(* IEC 61131-3 sources: ServoDriveControllerCode_Gen3SOScompressor/src/FB, 18 files *)

(* ---- FB_AnalogInputFilter.st ---- *)
(* ============================================================================
   FB_AnalogInputFilter - Analog Input Filter with Median and Low-Pass

   Project: Gen3 SOS Compressor Servo Controller
   Controller: Yaskawa MP2600iec

   Description:
   Two-stage analog input filter:
   1. Median filter (size 3 or 5) - Removes spike noise and outliers
   2. Low-pass filter (first-order IIR) - Smooths signal, configured by alpha

   The median filter runs first to remove impulsive noise, then the low-pass
   filter smooths the result. This combination is effective for industrial
   analog signals that may have both spike noise and high-frequency interference.

   Low-pass filter implementation:
   - First-order IIR: y[n] = alpha * x[n] + (1-alpha) * y[n-1]
   - Alpha should be calculated by caller: alpha = dt / (tau + dt)
   - Where dt = task cycle time, tau = desired time constant
   - Higher alpha = faster response, less smoothing
   - Lower alpha = slower response, more smoothing

   Configuration:
   - Alpha: Filter coefficient (0.0-1.0), calculated in PRG_Main ST_INIT
   - MedianFilterSize: 3 or 5 samples for median filter
   ============================================================================ *)

FUNCTION_BLOCK FB_AnalogInputFilter
VAR_INPUT
    Enable              : BOOL := TRUE;     (* Enable filtering *)
    RawInput            : INT;              (* Raw analog input (-32768 to +32767) *)
    Alpha               : LREAL;            (* Low-pass filter coefficient (0.0-1.0) *)
    MedianFilterSize    : INT := 3;         (* Median filter size: 3 or 5 *)
END_VAR

VAR_OUTPUT
    FilteredOutput      : INT;              (* Filtered output value *)
    FilteredReal        : LREAL;            (* Filtered output as LREAL *)
    RawReal             : LREAL;            (* Raw input as LREAL *)
END_VAR

VAR
    (* Median filter buffer (size 5, use 3 or 5 based on config) *)
    aMedianBuffer       : ARRAY[0..4] OF LREAL;
    nMedianIndex        : INT := 0;
    aSortBuffer         : ARRAY[0..4] OF LREAL;

    (* Low-pass filter state *)
    rFilteredValue      : LREAL := 0.0;
    rAlpha              : LREAL;

    (* Initialization flag *)
    bInitialized        : BOOL := FALSE;

    (* Temporary variables *)
    i, j                : INT;
    rTemp               : LREAL;
    rMedianResult       : LREAL;
    nSize               : INT;
END_VAR

(* ============================================================================
   Main Logic
   ============================================================================ *)

IF NOT Enable THEN
    (* Pass through raw value when disabled *)
    RawReal := INT_TO_LREAL(RawInput);
    FilteredReal := RawReal;
    FilteredOutput := RawInput;
    RETURN;
END_IF

(* Convert raw input to LREAL *)
RawReal := INT_TO_LREAL(RawInput);

(* Clamp alpha to valid range *)
rAlpha := LIMIT(0.0, Alpha, 1.0);

(* --------------------------------------------------------------------------
   Initialization
   -------------------------------------------------------------------------- *)

IF NOT bInitialized THEN
    (* Fill median buffer with current value *)
    FOR i := 0 TO 4 DO
        aMedianBuffer[i] := RawReal;
    END_FOR
    rFilteredValue := RawReal;
    bInitialized := TRUE;
END_IF

(* --------------------------------------------------------------------------
   Stage 1: Median Filter
   -------------------------------------------------------------------------- *)

(* Limit median size to 3 or 5 *)
IF MedianFilterSize >= 5 THEN
    nSize := 5;
ELSE
    nSize := 3;
END_IF

(* Add new sample to circular buffer *)
aMedianBuffer[nMedianIndex] := RawReal;
nMedianIndex := nMedianIndex + 1;
IF nMedianIndex >= nSize THEN
    nMedianIndex := 0;
END_IF

(* Copy to sort buffer *)
FOR i := 0 TO nSize - 1 DO
    aSortBuffer[i] := aMedianBuffer[i];
END_FOR

(* Simple bubble sort (efficient for small arrays) *)
FOR i := 0 TO nSize - 2 DO
    FOR j := 0 TO nSize - 2 - i DO
        IF aSortBuffer[j] > aSortBuffer[j + 1] THEN
            rTemp := aSortBuffer[j];
            aSortBuffer[j] := aSortBuffer[j + 1];
            aSortBuffer[j + 1] := rTemp;
        END_IF
    END_FOR
END_FOR

(* Get median value (middle element) *)
rMedianResult := aSortBuffer[nSize / 2];

(* --------------------------------------------------------------------------
   Stage 2: Low-Pass Filter (First-Order IIR)
   -------------------------------------------------------------------------- *)

(* Apply low-pass filter: y[n] = alpha * x[n] + (1-alpha) * y[n-1] *)
rFilteredValue := (rAlpha * rMedianResult) + ((1.0 - rAlpha) * rFilteredValue);

(* --------------------------------------------------------------------------
   Output
   -------------------------------------------------------------------------- *)

FilteredReal := rFilteredValue;

(* Convert back to INT with clamping *)
IF rFilteredValue < -32768.0 THEN
    FilteredOutput := -32768;
ELSIF rFilteredValue > 32767.0 THEN
    FilteredOutput := 32767;
ELSE
    FilteredOutput := LREAL_TO_INT(rFilteredValue);
END_IF

END_FUNCTION_BLOCK

(* ---- FB_AnalogProcessor.st ---- *)
(* ============================================================================
   FB_AnalogProcessor - Analog I/O Scaling and Processing

   Project: Gen3 SOS Compressor Servo Controller
   Controller: Yaskawa MP2600iec

   Description:
   Handles scaling of analog input signals for position, velocity, and torque
   reference based on the current operating mode.

   Analog Input Scaling:
   - Raw INT: -32768 to +32767 corresponds to -10V to +10V
   - Scaled to engineering units based on mode and configuration

   Position Mode uses two-stage mapping for consistency with position feedback:
   - Stage 1: In-cylinder region (higher resolution)
   - Stage 2: Out-of-cylinder region (lower resolution)

   Modes:
   - Position (010): Scale to mm using two-stage mapping
   - Velocity (011): Scale to mm/s (linear)
   - Torque (100): Scale to % of rated torque (linear)
   ============================================================================ *)

FUNCTION_BLOCK FB_AnalogProcessor
VAR_INPUT
    Enable              : BOOL;             (* Enable the processor *)
    RawAnalogInput      : INT;              (* Raw analog input value *)
    CurrentMode         : E_OperatingMode;  (* Current operating mode *)

    (* Two-stage position scaling configuration (same as output mapping) *)
    Stage1PosMin        : LREAL;            (* Stage 1 position start (mm) *)
    Stage1PosMax        : LREAL;            (* Stage 1 position end (mm) = transition pos *)
    Stage1VoltMin       : LREAL;            (* Stage 1 voltage start (V) *)
    Stage1VoltMax       : LREAL;            (* Stage 1 voltage end (V) = transition volt *)
    Stage2PosMin        : LREAL;            (* Stage 2 position start (mm) = transition pos *)
    Stage2PosMax        : LREAL;            (* Stage 2 position end (mm) *)
    Stage2VoltMin       : LREAL;            (* Stage 2 voltage start (V) = transition volt *)
    Stage2VoltMax       : LREAL;            (* Stage 2 voltage end (V) *)

    (* Velocity scaling configuration *)
    VelMin              : LREAL;            (* Velocity at -10V (mm/s) *)
    VelMax              : LREAL;            (* Velocity at +10V (mm/s) *)

    (* Torque scaling configuration *)
    TorqueMin           : LREAL;            (* Torque at -10V (%) *)
    TorqueMax           : LREAL;            (* Torque at +10V (%) *)
END_VAR

VAR_OUTPUT
    ScaledPosition      : LREAL;            (* Scaled position reference (mm) *)
    ScaledVelocity      : LREAL;            (* Scaled velocity reference (mm/s) *)
    ScaledTorque        : LREAL;            (* Scaled torque reference (%) *)
    ActiveReference     : LREAL;            (* Currently active reference value *)
    NormalizedInput     : LREAL;            (* Input normalized to 0.0-1.0 range *)
    InputVoltage        : LREAL;            (* Calculated input voltage (-10 to +10) *)
    InStage1            : BOOL;             (* Position input is in stage 1 region *)
    InStage2            : BOOL;             (* Position input is in stage 2 region *)
END_VAR

VAR
    rNormalized         : LREAL;            (* Normalized value 0.0 to 1.0 *)
    rStageNormalized    : LREAL;            (* Normalized value within stage *)
END_VAR

(* ============================================================================
   Constants
   ============================================================================ *)
VAR CONSTANT
    RAW_MIN             : LREAL := -32768.0;    (* Minimum raw value *)
    RAW_MAX             : LREAL := 32767.0;     (* Maximum raw value *)
    RAW_RANGE           : LREAL := 65535.0;     (* Total raw range *)
    VOLT_MIN            : LREAL := -10.0;       (* Minimum voltage *)
    VOLT_MAX            : LREAL := 10.0;        (* Maximum voltage *)
    VOLT_RANGE          : LREAL := 20.0;        (* Total voltage range *)
END_VAR

(* ============================================================================
   Main Logic
   ============================================================================ *)

IF NOT Enable THEN
    ScaledPosition := 0.0;
    ScaledVelocity := 0.0;
    ScaledTorque := 0.0;
    ActiveReference := 0.0;
    NormalizedInput := 0.5;
    InputVoltage := 0.0;
    InStage1 := FALSE;
    InStage2 := FALSE;
    RETURN;
END_IF

(* Normalize raw input to 0.0-1.0 range *)
rNormalized := (INT_TO_LREAL(RawAnalogInput) - RAW_MIN) / RAW_RANGE;
NormalizedInput := rNormalized;

(* Calculate input voltage *)
InputVoltage := VOLT_MIN + (rNormalized * VOLT_RANGE);

(* Scale velocity and torque (simple linear mapping) *)
ScaledVelocity := VelMin + (rNormalized * (VelMax - VelMin));
ScaledTorque := TorqueMin + (rNormalized * (TorqueMax - TorqueMin));

(* Scale position using two-stage mapping (inverse of FB_PositionMapping) *)
(* Determine which stage based on input voltage *)
(* Use < (not <=) so boundary value is handled by stage 2 only *)
IF InputVoltage < Stage1VoltMax THEN
    (* Stage 1: In-cylinder region *)
    InStage1 := TRUE;
    InStage2 := FALSE;

    (* Calculate normalized position within stage 1 *)
    IF (Stage1VoltMax - Stage1VoltMin) > 0.0 THEN
        rStageNormalized := (InputVoltage - Stage1VoltMin) / (Stage1VoltMax - Stage1VoltMin);
    ELSE
        rStageNormalized := 0.0;
    END_IF

    (* Clamp to 0.0-1.0 range *)
    rStageNormalized := LIMIT(0.0, rStageNormalized, 1.0);

    (* Calculate position for stage 1 *)
    ScaledPosition := Stage1PosMin + (rStageNormalized * (Stage1PosMax - Stage1PosMin));

ELSE
    (* Stage 2: Out-of-cylinder region *)
    InStage1 := FALSE;
    InStage2 := TRUE;

    (* Calculate normalized position within stage 2 *)
    IF (Stage2VoltMax - Stage2VoltMin) > 0.0 THEN
        rStageNormalized := (InputVoltage - Stage2VoltMin) / (Stage2VoltMax - Stage2VoltMin);
    ELSE
        rStageNormalized := 0.0;
    END_IF

    (* Clamp to 0.0-1.0 range *)
    rStageNormalized := LIMIT(0.0, rStageNormalized, 1.0);

    (* Calculate position for stage 2 *)
    ScaledPosition := Stage2PosMin + (rStageNormalized * (Stage2PosMax - Stage2PosMin));
END_IF

(* Select active reference based on mode *)
CASE CurrentMode OF
    MODE_POSITION:
        ActiveReference := ScaledPosition;

    MODE_VELOCITY:
        ActiveReference := ScaledVelocity;

    MODE_TORQUE:
        ActiveReference := ScaledTorque;

ELSE
    ActiveReference := 0.0;
END_CASE

END_FUNCTION_BLOCK

(* ---- FB_DigitalInputFilter.st ---- *)
(* ============================================================================
   FB_DigitalInputFilter - Digital Input Debounce Filter

   Project: Gen3 SOS Compressor Servo Controller
   Controller: Yaskawa MP2600iec

   Description:
   Debounces a digital input signal by requiring the input to be stable for
   a configurable time before the output changes.

   Features:
   - Configurable debounce time
   - Edge detection outputs
   - Raw input passthrough for debugging
   ============================================================================ *)

FUNCTION_BLOCK FB_DigitalInputFilter
VAR_INPUT
    RawInput            : BOOL;             (* Raw digital input *)
    DebounceTime        : TIME := T#10MS;   (* Debounce time *)
END_VAR

VAR_OUTPUT
    FilteredOutput      : BOOL;             (* Debounced output *)
    RisingEdge          : BOOL;             (* Rising edge detected on filtered output *)
    FallingEdge         : BOOL;             (* Falling edge detected on filtered output *)
    Stable              : BOOL;             (* Output has been stable (not changing) *)
    RawPassthrough      : BOOL;             (* Raw input passthrough for debugging *)
END_VAR

VAR
    tDebounce           : TON;              (* Debounce timer *)
    bLastRaw            : BOOL;             (* Previous raw input state *)
    bLastFiltered       : BOOL;             (* Previous filtered output state *)
    bPendingState       : BOOL;             (* State we're debouncing toward *)
    bFirstScan          : BOOL := TRUE;     (* First scan flag for initialization *)
END_VAR

(* ============================================================================
   Main Logic
   ============================================================================ *)

(* Passthrough for debugging *)
RawPassthrough := RawInput;

(* First scan initialization - accept current input state immediately *)
IF bFirstScan THEN
    FilteredOutput := RawInput;
    bLastRaw := RawInput;
    bLastFiltered := RawInput;
    bPendingState := RawInput;
    Stable := TRUE;
    RisingEdge := FALSE;
    FallingEdge := FALSE;
    bFirstScan := FALSE;
    RETURN;
END_IF

(* Detect raw input change *)
IF RawInput <> bLastRaw THEN
    (* Input changed - start debouncing toward new state *)
    bPendingState := RawInput;
    tDebounce(IN := FALSE);  (* Reset timer *)
END_IF

bLastRaw := RawInput;

(* Run debounce timer if pending state differs from current output *)
IF bPendingState <> FilteredOutput THEN
    tDebounce(IN := TRUE, PT := DebounceTime);
    Stable := FALSE;

    IF tDebounce.Q THEN
        (* Debounce complete - update output *)
        FilteredOutput := bPendingState;
        tDebounce(IN := FALSE);
        Stable := TRUE;
    END_IF
ELSE
    (* No state change pending *)
    tDebounce(IN := FALSE);
    Stable := TRUE;
END_IF

(* Edge detection on filtered output *)
RisingEdge := FilteredOutput AND NOT bLastFiltered;
FallingEdge := NOT FilteredOutput AND bLastFiltered;
bLastFiltered := FilteredOutput;

END_FUNCTION_BLOCK

(* ---- FB_EncoderManager.st ---- *)
(* ============================================================================
   FB_EncoderManager - Absolute Encoder Validation Manager

   Project: Gen3 SOS Compressor Servo Controller
   Controller: Yaskawa MP2600iec

   Description:
   Validates absolute encoder status on startup using Yaskawa's
   AbsolutePositionManager function block. Determines if homing is required
   due to encoder battery failure or multi-turn data corruption.

   The Sigma-7 absolute encoder maintains position across power cycles via
   battery backup. If the battery fails or multi-turn data is corrupted,
   the encoder position is invalid and homing is required.

   States:
   - IDLE: Waiting for check trigger
   - CHECK_INIT: Initialize AbsolutePositionManager
   - CHECK_STATUS: Query encoder status
   - COMPLETE: Check finished, outputs valid
   - ERROR: Error during check

   Integration:
   - Called from ST_ENCODER_CHECK state in PRG_Main
   - Sets AbsHomeRequired output if encoder invalid
   - PRG_Main uses this to set flagAbsHomeRequired
   ============================================================================ *)

FUNCTION_BLOCK FB_EncoderManager
VAR_INPUT
    Enable              : BOOL;             (* Enable the function block *)
    Axis                : AXIS_REF;         (* PLCopen axis reference *)
    CheckOnStartup      : BOOL;             (* Trigger startup check *)
END_VAR

VAR_OUTPUT
    EncoderValid        : BOOL;             (* Absolute position is valid *)
    BatteryOK           : BOOL;             (* Encoder battery status OK *)
    MultiTurnValid      : BOOL;             (* Multi-turn counter data valid *)
    AbsHomeRequired     : BOOL;             (* Homing required due to encoder issue *)
    CheckComplete       : BOOL;             (* Startup check finished *)
    Busy                : BOOL;             (* Check in progress *)
    Error               : BOOL;             (* Error occurred during check *)
    ErrorID             : DWORD;            (* Error code if Error=TRUE *)
END_VAR

VAR
    (* Yaskawa AbsolutePositionManager function block *)
    fbAbsPosManager     : AbsolutePositionManager;

    (* State machine *)
    eState              : INT := ENC_IDLE;

    (* Edge detection *)
    rTrigCheck          : R_TRIG;

    (* Timeout *)
    tCheckTimeout       : TON;

    (* Internal status *)
    bCheckTriggered     : BOOL;
END_VAR

(* ============================================================================
   Constants
   ============================================================================ *)
VAR CONSTANT
    ENC_IDLE            : INT := 0;         (* Idle state *)
    ENC_CHECK_INIT      : INT := 1;         (* Initialize check *)
    ENC_CHECK_STATUS    : INT := 2;         (* Query status *)
    ENC_COMPLETE        : INT := 3;         (* Check complete *)
    ENC_ERROR           : INT := 4;         (* Error state *)

    CHECK_TIMEOUT       : TIME := T#2S;     (* Timeout for encoder check *)
END_VAR

(* ============================================================================
   Main Logic
   ============================================================================ *)

IF NOT Enable THEN
    (* Reset all outputs when disabled *)
    EncoderValid := FALSE;
    BatteryOK := FALSE;
    MultiTurnValid := FALSE;
    AbsHomeRequired := FALSE;
    CheckComplete := FALSE;
    Busy := FALSE;
    Error := FALSE;
    ErrorID := 0;
    eState := ENC_IDLE;
    tCheckTimeout(IN := FALSE);
    fbAbsPosManager(Enable := FALSE);
    RETURN;
END_IF

(* Detect rising edge on CheckOnStartup *)
rTrigCheck(CLK := CheckOnStartup);

CASE eState OF

    ENC_IDLE:
        (* Waiting for check trigger *)
        Busy := FALSE;
        CheckComplete := FALSE;

        IF rTrigCheck.Q OR (CheckOnStartup AND NOT bCheckTriggered) THEN
            bCheckTriggered := TRUE;
            Busy := TRUE;
            Error := FALSE;
            ErrorID := 0;
            tCheckTimeout(IN := FALSE);
            eState := ENC_CHECK_INIT;
        END_IF

    ENC_CHECK_INIT:
        (* Initialize AbsolutePositionManager *)
        (* Start timeout timer *)
        tCheckTimeout(IN := TRUE, PT := CHECK_TIMEOUT);

        (* Enable the AbsolutePositionManager *)
        fbAbsPosManager(
            Axis := Axis,
            Enable := TRUE
        );

        (* Wait for FB to initialize or check for immediate status *)
        IF fbAbsPosManager.Valid THEN
            eState := ENC_CHECK_STATUS;
        ELSIF fbAbsPosManager.Error THEN
            Error := TRUE;
            ErrorID := fbAbsPosManager.ErrorID;
            eState := ENC_ERROR;
        ELSIF tCheckTimeout.Q THEN
            Error := TRUE;
            ErrorID := 16#8001;  (* Timeout error code *)
            eState := ENC_ERROR;
        END_IF

    ENC_CHECK_STATUS:
        (* Query encoder status from AbsolutePositionManager *)
        fbAbsPosManager(
            Axis := Axis,
            Enable := TRUE
        );

        (* Read status outputs *)
        (* Note: Actual output names depend on Yaskawa's AbsolutePositionManager interface *)
        (* Common outputs: AbsolutePositionValid, BatteryStatus, etc. *)

        (* Check for valid absolute position *)
        IF fbAbsPosManager.Valid THEN
            (* Evaluate encoder health *)
            (* AbsolutePositionManager typically provides:
               - Valid: Overall validity
               - AbsolutePositionValid: Position data is valid
               - BatteryAlarm: Battery has failed or is low
               - MultiTurnOverflow: Multi-turn counter overflow *)

            (* For Sigma-7, check if position is valid and no alarms *)
            EncoderValid := fbAbsPosManager.AbsolutePositionValid;
            BatteryOK := NOT fbAbsPosManager.BatteryAlarm;
            MultiTurnValid := NOT fbAbsPosManager.MultiTurnOverflow;

            (* Homing required if any issue detected *)
            AbsHomeRequired := NOT EncoderValid OR
                               NOT BatteryOK OR
                               NOT MultiTurnValid;

            CheckComplete := TRUE;
            Busy := FALSE;
            tCheckTimeout(IN := FALSE);
            eState := ENC_COMPLETE;

        ELSIF fbAbsPosManager.Error THEN
            Error := TRUE;
            ErrorID := fbAbsPosManager.ErrorID;
            eState := ENC_ERROR;

        ELSIF tCheckTimeout.Q THEN
            Error := TRUE;
            ErrorID := 16#8001;  (* Timeout error code *)
            eState := ENC_ERROR;
        END_IF

    ENC_COMPLETE:
        (* Check complete - hold outputs until disabled or new check *)
        Busy := FALSE;
        CheckComplete := TRUE;

        (* Allow re-check if CheckOnStartup toggled *)
        IF NOT CheckOnStartup THEN
            bCheckTriggered := FALSE;
        END_IF

        IF rTrigCheck.Q THEN
            (* New check requested *)
            CheckComplete := FALSE;
            Busy := TRUE;
            tCheckTimeout(IN := FALSE);
            eState := ENC_CHECK_INIT;
        END_IF

    ENC_ERROR:
        (* Error state *)
        Busy := FALSE;
        CheckComplete := FALSE;

        (* Assume encoder invalid on error - safe default *)
        EncoderValid := FALSE;
        BatteryOK := FALSE;
        MultiTurnValid := FALSE;
        AbsHomeRequired := TRUE;

        (* Disable the AbsolutePositionManager *)
        fbAbsPosManager(Enable := FALSE);
        tCheckTimeout(IN := FALSE);

        (* Allow retry if CheckOnStartup toggled *)
        IF NOT CheckOnStartup THEN
            bCheckTriggered := FALSE;
            Error := FALSE;
            ErrorID := 0;
            eState := ENC_IDLE;
        END_IF

END_CASE

END_FUNCTION_BLOCK

(* ---- FB_GoHome.st ---- *)
(* ============================================================================
   FB_GoHome - Go Home Mode Handler (Mode 101)

   Project: Gen3 SOS Compressor Servo Controller
   Controller: Yaskawa MP2600iec

   Description:
   Handles Mode 101 (Go Home) which moves the axis to the home position
   (at the home limit switch). This mode checks homing requirements before
   executing and redirects to homing mode if needed.

   Behavior:
   - If AbsHomeRequired is TRUE: Set RedirectToHoming, PRG_Main switches to 110
   - If requirements met: Execute MC_MoveAbsolute to HomePosition
   - After reaching position: Hold there until mode change

   Note: EOTHomeRequired does NOT block Go Home - the axis can still move
   to the home position even if EOT homing hasn't been done. Only
   AbsHomeRequired (encoder validity) blocks the move.

   Integration:
   - Called from ST_GO_HOME state in PRG_Main
   - RedirectToHoming signals PRG_Main to switch to ST_HOME_LIMIT
   - Abort input for motion enable drop handling
   ============================================================================ *)

FUNCTION_BLOCK FB_GoHome
VAR_INPUT
    Enable              : BOOL;             (* Enable the function block *)
    Execute             : BOOL;             (* Start go home sequence *)
    Axis                : AXIS_REF;         (* PLCopen axis reference *)

    (* Homing requirement flags *)
    AbsHomeRequired     : BOOL;             (* Encoder homing required (blocks Go Home) *)
    EOTHomeRequired     : BOOL;             (* EOT homing required (does NOT block) *)

    (* Configuration *)
    HomePosition        : LREAL;            (* Target home position (mm) *)
    HomeVelocity        : LREAL;            (* Movement velocity (mm/s) *)

    (* Control *)
    Abort               : BOOL;             (* Abort the move *)
END_VAR

VAR_OUTPUT
    Active              : BOOL;             (* Sequence is running *)
    Done                : BOOL;             (* At home position *)
    AtPosition          : BOOL;             (* Currently at home position *)
    HomingRequired      : BOOL;             (* Homing must be done first *)
    RedirectToHoming    : BOOL;             (* Caller should switch to homing mode *)
    InMotion            : BOOL;             (* Currently moving *)
    Error               : BOOL;             (* Error occurred *)
    ErrorID             : DWORD;            (* Error code if Error=TRUE *)
END_VAR

VAR
    (* PLCopen function blocks *)
    fbMoveAbsolute      : MC_MoveAbsolute;
    fbHalt              : MC_Halt;

    (* State machine *)
    eState              : INT := GOH_IDLE;

    (* Edge detection *)
    rTrigExecute        : R_TRIG;

    (* Position tolerance for "at position" detection *)
    rPosTolerance       : LREAL := 0.1;     (* mm *)
END_VAR

(* ============================================================================
   Constants
   ============================================================================ *)
VAR CONSTANT
    GOH_IDLE            : INT := 0;         (* Idle state *)
    GOH_CHECK_REQ       : INT := 1;         (* Check requirements *)
    GOH_REDIRECT        : INT := 2;         (* Redirect to homing *)
    GOH_MOVING          : INT := 3;         (* Moving to home *)
    GOH_AT_POSITION     : INT := 4;         (* At home position *)
    GOH_ABORTING        : INT := 5;         (* Aborting move *)
    GOH_ERROR           : INT := 6;         (* Error state *)
END_VAR

(* ============================================================================
   Main Logic
   ============================================================================ *)

IF NOT Enable THEN
    (* Reset all outputs when disabled *)
    Active := FALSE;
    Done := FALSE;
    AtPosition := FALSE;
    HomingRequired := FALSE;
    RedirectToHoming := FALSE;
    InMotion := FALSE;
    Error := FALSE;
    ErrorID := 0;
    eState := GOH_IDLE;
    fbMoveAbsolute(Execute := FALSE);
    fbHalt(Execute := FALSE);
    RETURN;
END_IF

(* Detect rising edge on Execute *)
rTrigExecute(CLK := Execute);

(* Handle abort in any state *)
IF Abort AND (eState <> GOH_IDLE) AND (eState <> GOH_ERROR) AND (eState <> GOH_REDIRECT) THEN
    fbMoveAbsolute(Execute := FALSE);
    eState := GOH_ABORTING;
END_IF

CASE eState OF

    GOH_IDLE:
        (* Waiting for execute command *)
        Active := FALSE;
        Done := FALSE;
        AtPosition := FALSE;
        HomingRequired := FALSE;
        RedirectToHoming := FALSE;
        InMotion := FALSE;
        Error := FALSE;
        ErrorID := 0;

        (* Reset function blocks *)
        fbMoveAbsolute(Execute := FALSE);
        fbHalt(Execute := FALSE);

        IF rTrigExecute.Q OR Execute THEN
            Active := TRUE;
            eState := GOH_CHECK_REQ;
        END_IF

    GOH_CHECK_REQ:
        (* Check homing requirements *)

        IF AbsHomeRequired THEN
            (* Encoder homing required - cannot go home without valid position *)
            HomingRequired := TRUE;
            RedirectToHoming := TRUE;
            eState := GOH_REDIRECT;

        ELSE
            (* Requirements met (or only EOT homing needed) - proceed with move *)
            HomingRequired := FALSE;
            RedirectToHoming := FALSE;
            eState := GOH_MOVING;
        END_IF

    GOH_REDIRECT:
        (* Waiting for PRG_Main to handle redirect *)
        (* Stay in this state - PRG_Main will transition to ST_HOME_LIMIT *)
        (* This FB will be disabled when state changes *)
        Active := TRUE;
        HomingRequired := TRUE;
        RedirectToHoming := TRUE;

    GOH_MOVING:
        (* Execute move to home position *)
        fbMoveAbsolute(
            Axis := Axis,
            Execute := TRUE,
            Position := HomePosition,
            Velocity := HomeVelocity,
            Acceleration := 0.0,    (* Use axis default *)
            Deceleration := 0.0,    (* Use axis default *)
            Jerk := 0.0             (* Use axis default *)
        );

        InMotion := fbMoveAbsolute.Busy;

        IF fbMoveAbsolute.Done THEN
            (* Move complete - reset FB for next use
               NOTE: Setting Execute := FALSE does NOT release position control.
               Per PLCopen standard, axis remains in "Standstill" state with
               active servo position holding. This is standard practice. *)
            fbMoveAbsolute(Execute := FALSE);
            Done := TRUE;
            AtPosition := TRUE;
            InMotion := FALSE;
            eState := GOH_AT_POSITION;

        ELSIF fbMoveAbsolute.Error THEN
            (* Move failed *)
            Error := TRUE;
            ErrorID := fbMoveAbsolute.ErrorID;
            fbMoveAbsolute(Execute := FALSE);
            eState := GOH_ERROR;

        ELSIF fbMoveAbsolute.CommandAborted THEN
            (* Move was aborted externally *)
            fbMoveAbsolute(Execute := FALSE);
            eState := GOH_ABORTING;
        END_IF

    GOH_AT_POSITION:
        (* At home position - hold here until mode change *)
        Done := TRUE;
        AtPosition := TRUE;
        InMotion := FALSE;
        Active := TRUE;

        (* Check if still at position (could drift in some cases) *)
        (* Note: In practice, the drive holds position in servo mode *)

        (* If Execute goes low, we can reset for next time *)
        IF NOT Execute THEN
            Done := FALSE;
            eState := GOH_IDLE;
        END_IF

    GOH_ABORTING:
        (* Aborting move - execute halt *)
        fbHalt(
            Axis := Axis,
            Execute := TRUE
        );

        IF fbHalt.Done THEN
            fbHalt(Execute := FALSE);
            Active := FALSE;
            InMotion := FALSE;
            eState := GOH_IDLE;

        ELSIF fbHalt.Error THEN
            (* Halt failed - still try to go to idle *)
            fbHalt(Execute := FALSE);
            eState := GOH_ERROR;
        END_IF

    GOH_ERROR:
        (* Error state *)
        Active := FALSE;
        InMotion := FALSE;
        Done := FALSE;

        (* Allow reset when Execute goes low *)
        IF NOT Execute THEN
            Error := FALSE;
            ErrorID := 0;
            eState := GOH_IDLE;
        END_IF

END_CASE

END_FUNCTION_BLOCK

(* ---- FB_HandshakeManager.st ---- *)
(* ============================================================================
   FB_HandshakeManager - Master-Slave Handshake Manager

   Project: Gen3 SOS Compressor Servo Controller
   Controller: Yaskawa MP2600iec

   Description:
   Manages the handshake protocol between master and slave for:
   1. Mode entry handshake: 3-bit mode command/confirmation with timeout
   2. Fault reset handshake: FaultReset HIGH + MotionEnable LOW + fault mirroring

   Mode Entry Handshake Sequence:
   1. Master sets mode bits (DI0-2)
   2. Slave decodes and validates mode
   3. Slave sets confirmation bits (DO0-2) to match
   4. Master sets diMotionEnable HIGH
   5. Slave verifies mode bits still match → handshake complete
   6. If timeout or mismatch → handshake failed

   Fault Reset Handshake (with fault code mirroring):
   1. Slave is in fault state with doFaultActive = HIGH
   2. Slave outputs fault code on DO0-DO2
   3. Master reads fault code and sets DI0-DI2 to mirror it
   4. Master sets diFaultReset HIGH while diMotionEnable = LOW
   5. Slave verifies DI0-DI2 matches fault code (level-based, not edge)
   6. FaultResetValid goes TRUE, caller clears fault
   7. Master sees fault cleared, releases diFaultReset

   NOTE: All inputs should be pre-filtered/debounced by the caller.
   ============================================================================ *)

FUNCTION_BLOCK FB_HandshakeManager
VAR_INPUT
    Enable              : BOOL;             (* Enable handshake manager *)

    (* Mode handshake inputs *)
    RequestedMode       : E_OperatingMode;  (* Mode requested by master *)
    ModeStable          : BOOL;             (* Mode inputs are stable *)
    MotionEnable        : BOOL;             (* Motion enable from master - should be filtered *)

    (* Fault reset inputs *)
    FaultReset          : BOOL;             (* Fault reset signal from master - should be filtered *)
    InFaultState        : BOOL;             (* Currently in fault state *)
    ActiveFaultCode     : E_FaultCode;      (* Active fault code for mirroring check *)

    (* Configuration *)
    HandshakeTimeout    : TIME := T#500MS;  (* Timeout for handshake *)
END_VAR

VAR_OUTPUT
    (* Mode handshake outputs *)
    ConfirmedMode       : E_OperatingMode;  (* Current confirmed mode (valid when HandshakeComplete) *)
    HandshakeActive     : BOOL;             (* TRUE from handshake start until complete/timeout *)
    HandshakeComplete   : BOOL;             (* TRUE when handshake succeeded (persists until MotionEnable drops) *)
    HandshakeTimeout_Q  : BOOL;             (* TRUE when timeout occurred (persists until MotionEnable drops) *)

    (* Confirmation bits for digital outputs *)
    ConfirmBit0         : BOOL;             (* DO0 value *)
    ConfirmBit1         : BOOL;             (* DO1 value *)
    ConfirmBit2         : BOOL;             (* DO2 value *)

    (* Fault reset outputs *)
    FaultResetEdge      : BOOL;             (* Fault reset rising edge detected (single scan pulse) *)
    FaultResetValid     : BOOL;             (* Fault reset conditions met (level-based, stays TRUE while valid) *)
END_VAR

VAR
    (* State machine *)
    eState              : INT := HS_IDLE;   (* Handshake state - initialized to HS_IDLE *)

    (* Timers *)
    tTimeout            : TON;              (* Handshake timeout timer *)

    (* Edge detection *)
    rTrigFaultReset     : R_TRIG;           (* Rising edge on fault reset *)

    (* Internal tracking *)
    eModeAtStart        : E_OperatingMode;  (* Mode when handshake started *)
    bModeStableAtStart  : BOOL;             (* Capture mode stability at handshake start *)
END_VAR

(* ============================================================================
   Constants for state machine
   ============================================================================ *)
VAR CONSTANT
    HS_IDLE             : INT := 0;         (* Idle, no handshake active *)
    HS_WAIT_MOTION_EN   : INT := 1;         (* Waiting for motion enable *)
    HS_VERIFY_MODE      : INT := 2;         (* Verifying mode match *)
    HS_COMPLETE         : INT := 3;         (* Handshake complete *)
    HS_TIMEOUT          : INT := 4;         (* Handshake timed out *)
END_VAR

(* ============================================================================
   Main Logic
   ============================================================================ *)

IF NOT Enable THEN
    (* Reset all outputs when disabled *)
    ConfirmedMode := MODE_IDLE;
    HandshakeActive := FALSE;
    HandshakeComplete := FALSE;
    HandshakeTimeout_Q := FALSE;
    ConfirmBit0 := FALSE;
    ConfirmBit1 := FALSE;
    ConfirmBit2 := FALSE;
    FaultResetEdge := FALSE;
    FaultResetValid := FALSE;
    eState := HS_IDLE;
    tTimeout(IN := FALSE);
    RETURN;
END_IF

(* --------------------------------------------------------------------------
   Fault Reset Handshake Detection (with fault code mirroring)
   Uses LEVEL-based detection to avoid race conditions.
   The caller should detect the rising edge of FaultResetValid if needed.
   -------------------------------------------------------------------------- *)
rTrigFaultReset(CLK := FaultReset);
FaultResetEdge := rTrigFaultReset.Q;

(* Fault reset is valid when ALL conditions are met (level-based):
   - FaultReset is HIGH (level, not edge)
   - MotionEnable is LOW
   - We are in fault state
   - Active fault code is not FAULT_NONE
   - Master has mirrored the fault code on DI0-2 (RequestedMode matches ActiveFaultCode) *)
FaultResetValid := FaultReset AND
                   (NOT MotionEnable) AND
                   InFaultState AND
                   (ActiveFaultCode <> FAULT_NONE) AND
                   FaultMatchesModeBits(ActiveFaultCode, RequestedMode);

(* --------------------------------------------------------------------------
   Mode Handshake State Machine
   -------------------------------------------------------------------------- *)
CASE eState OF

    HS_IDLE:
        (* Reset outputs *)
        HandshakeActive := FALSE;
        HandshakeComplete := FALSE;
        HandshakeTimeout_Q := FALSE;
        tTimeout(IN := FALSE);

        (* Start handshake when mode is stable and different from idle
           (or when transitioning to a new mode) *)
        IF ModeStable AND (RequestedMode <> MODE_IDLE) AND NOT MotionEnable THEN
            (* Set confirmation to match requested mode *)
            ConfirmedMode := RequestedMode;
            SetConfirmBits(RequestedMode);
            eModeAtStart := RequestedMode;
            bModeStableAtStart := TRUE;
            HandshakeActive := TRUE;
            eState := HS_WAIT_MOTION_EN;
            tTimeout(IN := TRUE, PT := HandshakeTimeout);
        ELSIF ModeStable AND (RequestedMode = MODE_IDLE) THEN
            (* Idle mode - just confirm it *)
            ConfirmedMode := MODE_IDLE;
            SetConfirmBits(MODE_IDLE);
        END_IF

    HS_WAIT_MOTION_EN:
        (* Waiting for master to assert motion enable *)
        (* Timer must be called each scan to update *)
        tTimeout(IN := TRUE, PT := HandshakeTimeout);

        IF tTimeout.Q THEN
            (* Timeout - handshake failed *)
            tTimeout(IN := FALSE);
            eState := HS_TIMEOUT;

        ELSIF RequestedMode <> eModeAtStart THEN
            (* Mode changed during handshake - abort and reset timer *)
            tTimeout(IN := FALSE);
            eState := HS_IDLE;

        ELSIF MotionEnable THEN
            (* Motion enable received, verify mode still matches *)
            eState := HS_VERIFY_MODE;
        END_IF

    HS_VERIFY_MODE:
        (* Verify requested mode hasn't changed since handshake start *)
        IF RequestedMode = eModeAtStart THEN
            (* Mode matches - handshake complete *)
            HandshakeComplete := TRUE;
            HandshakeActive := FALSE;
            tTimeout(IN := FALSE);
            eState := HS_COMPLETE;
        ELSE
            (* Mismatch - treat as timeout/failure *)
            tTimeout(IN := FALSE);
            eState := HS_TIMEOUT;
        END_IF

    HS_COMPLETE:
        (* Handshake complete - stay here until motion enable drops *)
        IF NOT MotionEnable THEN
            (* Motion disabled - return to idle *)
            HandshakeComplete := FALSE;
            eState := HS_IDLE;
        END_IF

    HS_TIMEOUT:
        (* Handshake timed out or failed *)
        HandshakeTimeout_Q := TRUE;
        HandshakeActive := FALSE;
        ConfirmedMode := MODE_IDLE;  (* Reset confirmed mode on failure *)
        SetConfirmBits(MODE_IDLE);
        tTimeout(IN := FALSE);

        (* Exit timeout when motion enable drops - simpler and more reliable *)
        IF NOT MotionEnable THEN
            HandshakeTimeout_Q := FALSE;
            eState := HS_IDLE;
        END_IF

END_CASE

END_FUNCTION_BLOCK

(* ============================================================================
   Helper Method: Set Confirmation Bits from Mode
   Uses centralized conversion functions from EnumConversions.st
   ============================================================================ *)
METHOD PRIVATE SetConfirmBits
VAR_INPUT
    Mode : E_OperatingMode;
END_VAR

(* Use centralized ModeToBits function *)
ModeToBits(Mode, ConfirmBit0, ConfirmBit1, ConfirmBit2);

END_METHOD

(* ---- FB_HomeEOT.st ---- *)
(* ============================================================================
   FB_HomeEOT - End-of-Travel Homing Sequence Handler (Mode 111)

   Project: Gen3 SOS Compressor Servo Controller
   Controller: Yaskawa MP2600iec

   Description:
   Encapsulates the complete End-of-Travel (EOT) homing sequence for Mode 111.
   Uses torque-limited velocity control to find the mechanical end stop, then
   calculates a coordinate offset for master/slave translation.

   Sequence:
   1. CHECK_REQ: Verify AbsHomeRequired is FALSE (limit switch homing must be done first)
   2. FAST_APPROACH: Fast jog toward EOT with torque limiting for safety
   3. SLOW_APPROACH: Slow torque-limited approach when near expected position
   4. STALL_DETECT: Confirm stall condition (velocity near zero, torque at limit)
   5. SETREF: Calculate coordinate offset (preserves encoder zero from Mode 110)

   Coordinate System:
   This FB calculates EOTOffset for master/slave coordinate transformation:
   - Master position = Slave position + EOTOffset
   - EOTOffset = ExpectedEOTPosition - ActualEOTPosition (encoder value at stall)

   This preserves the limit switch zero reference from Mode 110 while allowing
   the master to see the expected position value at EOT.

   Uses Y_DirectControl:
   - Mode 2 (velocity mode) with torque limiting for safe mechanical contact

   Integration:
   - Called from ST_HOME_EOT state in PRG_Main
   - RequiresLimitHome output signals need for Mode 110 first
   - Abort input for motion enable drop handling
   ============================================================================ *)

FUNCTION_BLOCK FB_HomeEOT
VAR_INPUT
    Enable              : BOOL;             (* Enable the function block *)
    Execute             : BOOL;             (* Start homing sequence *)
    Axis                : AXIS_REF;         (* PLCopen axis reference *)

    (* Homing requirement check *)
    AbsHomeRequired     : BOOL;             (* Limit switch homing required (blocks EOT homing) *)

    (* Configuration *)
    FastVelocity        : LREAL;            (* Fast approach velocity (mm/s) *)
    SlowVelocity        : LREAL;            (* Slow approach velocity (mm/s) *)
    TorqueLimit         : LREAL;            (* Torque limit during approach (%) *)
    TorqueThreshold     : LREAL;            (* Torque threshold for stall detection (%) *)
    ApproachDistance    : LREAL;            (* Distance before EOT to switch to slow (mm) *)
    ExpectedEOTPosition : LREAL;            (* Expected position at EOT (mm) *)
    StallDetectTime     : TIME;             (* Time to confirm stall condition *)
    Timeout             : TIME;             (* Overall sequence timeout *)

    (* Feedback inputs *)
    ActualPosition      : LREAL;            (* Current position (mm) *)
    ActualVelocity      : LREAL;            (* Current velocity (mm/s) *)
    ActualTorque        : LREAL;            (* Current torque (% of rated) *)

    (* Control *)
    Abort               : BOOL;             (* Abort the sequence *)
END_VAR

VAR_OUTPUT
    Active              : BOOL;             (* Sequence is running *)
    Done                : BOOL;             (* Homing complete *)
    InMotion            : BOOL;             (* Currently moving *)
    Error               : BOOL;             (* Error occurred *)
    ErrorID             : DWORD;            (* Error code if Error=TRUE *)
    RequiresLimitHome   : BOOL;             (* Must do limit switch homing first *)
    EOTPosition         : LREAL;            (* Recorded encoder position at EOT stall *)
    EOTOffset           : LREAL;            (* Calculated coordinate offset *)
END_VAR

VAR
    (* Yaskawa function blocks *)
    fbDirectControl     : Y_DirectControl;
    fbHalt              : MC_Halt;

    (* State machine *)
    eState              : INT := HE_IDLE;

    (* Edge detection *)
    rTrigExecute        : R_TRIG;

    (* Timers *)
    tTimeout            : TON;              (* Overall timeout *)
    tStallConfirm       : TON;              (* Stall confirmation timer *)

    (* Stall detection threshold with hysteresis *)
    rVelocityThreshold  : LREAL := 0.5;     (* mm/s - velocity considered "stopped" *)
    rTorqueMultiplier   : LREAL := 0.9;     (* Multiplier for torque threshold *)
END_VAR

(* ============================================================================
   Constants
   ============================================================================ *)
VAR CONSTANT
    HE_IDLE             : INT := 0;         (* Idle state *)
    HE_CHECK_REQ        : INT := 1;         (* Check requirements *)
    HE_REQUIRES_HOME    : INT := 2;         (* Limit homing required first *)
    HE_FAST_APPROACH    : INT := 3;         (* Fast approach to near EOT *)
    HE_SLOW_APPROACH    : INT := 4;         (* Slow torque-limited approach *)
    HE_STALL_DETECT     : INT := 5;         (* Confirming stall condition *)
    HE_SETREF           : INT := 6;         (* Calculate offset *)
    HE_DONE             : INT := 7;         (* Sequence complete *)
    HE_ABORTING         : INT := 8;         (* Aborting sequence *)
    HE_ERROR            : INT := 9;         (* Error state *)

    (* Error codes *)
    ERR_TIMEOUT         : DWORD := 16#8011; (* Homing timeout *)
    ERR_DRIVE           : DWORD := 16#8012; (* Drive error during homing *)
    ERR_LIMIT_REQ       : DWORD := 16#8013; (* Limit switch homing required *)
END_VAR

(* ============================================================================
   Main Logic
   ============================================================================ *)

IF NOT Enable THEN
    (* Reset all outputs when disabled *)
    Active := FALSE;
    Done := FALSE;
    InMotion := FALSE;
    Error := FALSE;
    ErrorID := 0;
    RequiresLimitHome := FALSE;
    EOTPosition := 0.0;
    EOTOffset := 0.0;
    eState := HE_IDLE;
    fbDirectControl(Enable := FALSE);
    fbHalt(Execute := FALSE);
    tTimeout(IN := FALSE);
    tStallConfirm(IN := FALSE);
    RETURN;
END_IF

(* Detect rising edge on Execute *)
rTrigExecute(CLK := Execute);

(* Handle abort in most states *)
IF Abort AND (eState <> HE_IDLE) AND (eState <> HE_ERROR) AND
   (eState <> HE_DONE) AND (eState <> HE_REQUIRES_HOME) THEN
    fbDirectControl(Enable := FALSE);
    tTimeout(IN := FALSE);
    tStallConfirm(IN := FALSE);
    eState := HE_ABORTING;
END_IF

(* Overall timeout check *)
tTimeout(IN := (eState >= HE_FAST_APPROACH) AND (eState <= HE_SETREF),
         PT := Timeout);

IF tTimeout.Q THEN
    fbDirectControl(Enable := FALSE);
    fbHalt(Execute := FALSE);
    Error := TRUE;
    ErrorID := ERR_TIMEOUT;
    eState := HE_ERROR;
END_IF

CASE eState OF

    HE_IDLE:
        (* Waiting for execute command *)
        Active := FALSE;
        Done := FALSE;
        InMotion := FALSE;
        Error := FALSE;
        ErrorID := 0;
        RequiresLimitHome := FALSE;
        EOTPosition := 0.0;
        EOTOffset := 0.0;

        (* Reset function blocks *)
        fbDirectControl(Enable := FALSE);
        fbHalt(Execute := FALSE);
        tTimeout(IN := FALSE);
        tStallConfirm(IN := FALSE);

        IF rTrigExecute.Q OR Execute THEN
            Active := TRUE;
            eState := HE_CHECK_REQ;
        END_IF

    HE_CHECK_REQ:
        (* Check if limit switch homing is required first *)
        IF AbsHomeRequired THEN
            (* Must do limit switch homing before EOT homing *)
            RequiresLimitHome := TRUE;
            eState := HE_REQUIRES_HOME;
        ELSE
            (* Requirements met - proceed to fast approach *)
            RequiresLimitHome := FALSE;
            eState := HE_FAST_APPROACH;
        END_IF

    HE_REQUIRES_HOME:
        (* Waiting for caller to handle the requirement *)
        (* PRG_Main should transition to fault or Mode 110 *)
        Active := TRUE;
        RequiresLimitHome := TRUE;
        (* Note: Caller should disable this FB and handle the error *)

    HE_FAST_APPROACH:
        (* Fast jog toward EOT (positive/extend direction) with torque limit *)
        fbDirectControl(
            Axis := Axis,
            Enable := TRUE,
            Mode := 2,  (* Velocity mode *)
            Velocity := FastVelocity,
            Torque := TorqueLimit
        );

        InMotion := fbDirectControl.InOperation;

        (* Switch to slow approach when near expected EOT *)
        IF ActualPosition >= (ExpectedEOTPosition - ApproachDistance) THEN
            fbDirectControl(Enable := FALSE);
            eState := HE_SLOW_APPROACH;

        ELSIF fbDirectControl.Error THEN
            fbDirectControl(Enable := FALSE);
            Error := TRUE;
            ErrorID := ERR_DRIVE;
            eState := HE_ERROR;
        END_IF

    HE_SLOW_APPROACH:
        (* Slow torque-limited approach to EOT *)
        fbDirectControl(
            Axis := Axis,
            Enable := TRUE,
            Mode := 2,  (* Velocity mode *)
            Velocity := SlowVelocity,
            Torque := TorqueLimit
        );

        InMotion := TRUE;
        tStallConfirm(IN := FALSE);  (* Reset stall timer *)

        (* Detect stall: velocity near zero while torque at limit *)
        IF (ABS(ActualVelocity) < rVelocityThreshold) AND
           (ABS(ActualTorque) >= TorqueThreshold * rTorqueMultiplier) THEN
            (* Stall condition detected - move to confirm *)
            eState := HE_STALL_DETECT;

        ELSIF fbDirectControl.Error THEN
            fbDirectControl(Enable := FALSE);
            Error := TRUE;
            ErrorID := ERR_DRIVE;
            eState := HE_ERROR;
        END_IF

    HE_STALL_DETECT:
        (* Confirm stall condition for StallDetectTime *)
        (* Continue pushing against EOT to confirm *)
        fbDirectControl(
            Axis := Axis,
            Enable := TRUE,
            Mode := 2,
            Velocity := SlowVelocity,
            Torque := TorqueLimit
        );

        InMotion := TRUE;

        (* Timer for stall confirmation *)
        tStallConfirm(IN := TRUE, PT := StallDetectTime);

        (* Check if still stalled *)
        IF (ABS(ActualVelocity) < rVelocityThreshold) AND
           (ABS(ActualTorque) >= TorqueThreshold * rTorqueMultiplier) THEN
            IF tStallConfirm.Q THEN
                (* Stall confirmed - proceed to set reference *)
                fbDirectControl(Enable := FALSE);
                eState := HE_SETREF;
            END_IF
        ELSE
            (* Not stalled anymore - go back to slow approach *)
            tStallConfirm(IN := FALSE);
            eState := HE_SLOW_APPROACH;
        END_IF

    HE_SETREF:
        (* Calculate EOT offset - DO NOT call MC_SetPosition
           This preserves the limit switch zero reference from Mode 110 *)

        (* First halt to ensure fully stopped *)
        fbHalt(
            Axis := Axis,
            Execute := NOT fbHalt.Done
        );

        IF fbHalt.Done THEN
            fbHalt(Execute := FALSE);

            (* Record actual encoder position at EOT stall *)
            EOTPosition := ActualPosition;

            (* Calculate offset for coordinate transformation *)
            (* Master position = Slave position + offset *)
            (* Example: If actual EOT is at encoder 295mm and expected is 300mm, *)
            (*          offset = 300 - 295 = 5mm *)
            (*          Master sees 300mm, slave is at 295mm *)
            EOTOffset := ExpectedEOTPosition - EOTPosition;

            InMotion := FALSE;
            Done := TRUE;
            eState := HE_DONE;
        END_IF

    HE_DONE:
        (* Homing sequence complete *)
        Done := TRUE;
        Active := TRUE;
        InMotion := FALSE;

        (* Reset when Execute goes low *)
        IF NOT Execute THEN
            Done := FALSE;
            eState := HE_IDLE;
        END_IF

    HE_ABORTING:
        (* Aborting sequence - halt motion *)
        fbDirectControl(Enable := FALSE);
        fbHalt(
            Axis := Axis,
            Execute := TRUE
        );

        IF fbHalt.Done THEN
            fbHalt(Execute := FALSE);
            Active := FALSE;
            InMotion := FALSE;
            eState := HE_IDLE;

        ELSIF fbHalt.Error THEN
            (* Halt failed - still try to go to idle *)
            fbHalt(Execute := FALSE);
            eState := HE_ERROR;
        END_IF

    HE_ERROR:
        (* Error state *)
        Active := FALSE;
        InMotion := FALSE;
        Done := FALSE;
        fbDirectControl(Enable := FALSE);

        (* Allow reset when Execute goes low *)
        IF NOT Execute THEN
            Error := FALSE;
            ErrorID := 0;
            eState := HE_IDLE;
        END_IF

END_CASE

END_FUNCTION_BLOCK

(* ---- FB_HomeLimit.st ---- *)
(* ============================================================================
   FB_HomeLimit - Limit Switch Homing Sequence Handler (Mode 110)

   Project: Gen3 SOS Compressor Servo Controller
   Controller: Yaskawa MP2600iec

   Description:
   Encapsulates the complete limit switch homing sequence for Mode 110.
   This FB handles the entire sequence from approach to setting the position
   reference, including over-travel detection and direction reversal.

   Sequence:
   1. APPROACH: Move toward home limit switch (negative direction first)
      - If retract limit triggers instead, reverse to positive direction
   2. DETECT: Halt motion when home limit switch detected
   3. BACKOFF: Move away from switch at slow speed until switch clears
   4. SETREF: Set position reference at switch edge location

   Over-Travel Handling:
   - If retract limit triggers during approach from negative direction,
     the FB automatically reverses to approach from positive direction
   - If retract limit triggers during positive approach, this is a fault

   Integration:
   - Called from ST_HOME_LIMIT state in PRG_Main
   - Abort input for motion enable drop handling
   ============================================================================ *)

FUNCTION_BLOCK FB_HomeLimit
VAR_INPUT
    Enable              : BOOL;             (* Enable the function block *)
    Execute             : BOOL;             (* Start homing sequence *)
    Axis                : AXIS_REF;         (* PLCopen axis reference *)

    (* Configuration *)
    ApproachVelocity    : LREAL;            (* Approach velocity (mm/s) *)
    BackoffVelocity     : LREAL;            (* Backoff velocity (mm/s) *)
    SetPosition         : LREAL;            (* Position to set at home switch (mm) *)
    Timeout             : TIME;             (* Overall sequence timeout *)

    (* Limit switch inputs *)
    LimitHomeActive     : BOOL;             (* Home limit switch is triggered *)
    LimitRetractActive  : BOOL;             (* Retract limit switch is triggered *)

    (* Control *)
    Abort               : BOOL;             (* Abort the sequence *)
END_VAR

VAR_OUTPUT
    Active              : BOOL;             (* Sequence is running *)
    Done                : BOOL;             (* Homing complete *)
    InMotion            : BOOL;             (* Currently moving *)
    Error               : BOOL;             (* Error occurred *)
    ErrorID             : DWORD;            (* Error code if Error=TRUE *)
    ApproachingPositive : BOOL;             (* Currently approaching from positive direction *)
END_VAR

VAR
    (* PLCopen function blocks *)
    fbMoveVelocity      : MC_MoveVelocity;
    fbHalt              : MC_Halt;
    fbSetPosition       : MC_SetPosition;

    (* State machine *)
    eState              : INT := HL_IDLE;

    (* Edge detection *)
    rTrigExecute        : R_TRIG;

    (* Timers *)
    tTimeout            : TON;

    (* Internal flags *)
    bApproachFromPositive : BOOL := FALSE;  (* Direction flag for over-travel handling *)
END_VAR

(* ============================================================================
   Constants
   ============================================================================ *)
VAR CONSTANT
    HL_IDLE             : INT := 0;         (* Idle state *)
    HL_APPROACH         : INT := 1;         (* Approaching limit switch *)
    HL_DETECT           : INT := 2;         (* Halt after limit detected *)
    HL_BACKOFF          : INT := 3;         (* Backing off from switch *)
    HL_SETREF           : INT := 4;         (* Setting position reference *)
    HL_DONE             : INT := 5;         (* Sequence complete *)
    HL_ABORTING         : INT := 6;         (* Aborting sequence *)
    HL_ERROR            : INT := 7;         (* Error state *)

    (* Error codes *)
    ERR_TIMEOUT         : DWORD := 16#8001; (* Homing timeout *)
    ERR_DRIVE           : DWORD := 16#8002; (* Drive error during homing *)
    ERR_LIMIT_INVALID   : DWORD := 16#8003; (* Invalid limit switch sequence *)
    ERR_SETPOS          : DWORD := 16#8004; (* Set position failed *)
END_VAR

(* ============================================================================
   Main Logic
   ============================================================================ *)

IF NOT Enable THEN
    (* Reset all outputs when disabled *)
    Active := FALSE;
    Done := FALSE;
    InMotion := FALSE;
    Error := FALSE;
    ErrorID := 0;
    ApproachingPositive := FALSE;
    eState := HL_IDLE;
    bApproachFromPositive := FALSE;
    fbMoveVelocity(Execute := FALSE);
    fbHalt(Execute := FALSE);
    fbSetPosition(Execute := FALSE);
    tTimeout(IN := FALSE);
    RETURN;
END_IF

(* Detect rising edge on Execute *)
rTrigExecute(CLK := Execute);

(* Handle abort in most states *)
IF Abort AND (eState <> HL_IDLE) AND (eState <> HL_ERROR) AND (eState <> HL_DONE) THEN
    fbMoveVelocity(Execute := FALSE);
    fbSetPosition(Execute := FALSE);
    tTimeout(IN := FALSE);
    eState := HL_ABORTING;
END_IF

(* Overall timeout check *)
tTimeout(IN := (eState <> HL_IDLE) AND (eState <> HL_DONE) AND (eState <> HL_ERROR) AND (eState <> HL_ABORTING),
         PT := Timeout);

IF tTimeout.Q THEN
    fbMoveVelocity(Execute := FALSE);
    fbHalt(Execute := FALSE);
    fbSetPosition(Execute := FALSE);
    Error := TRUE;
    ErrorID := ERR_TIMEOUT;
    eState := HL_ERROR;
END_IF

CASE eState OF

    HL_IDLE:
        (* Waiting for execute command *)
        Active := FALSE;
        Done := FALSE;
        InMotion := FALSE;
        Error := FALSE;
        ErrorID := 0;
        ApproachingPositive := FALSE;
        bApproachFromPositive := FALSE;

        (* Reset function blocks *)
        fbMoveVelocity(Execute := FALSE);
        fbHalt(Execute := FALSE);
        fbSetPosition(Execute := FALSE);
        tTimeout(IN := FALSE);

        IF rTrigExecute.Q OR Execute THEN
            Active := TRUE;
            bApproachFromPositive := FALSE;  (* Start approaching from negative *)
            eState := HL_APPROACH;
        END_IF

    HL_APPROACH:
        (* Move toward home limit switch
           Direction depends on bApproachFromPositive:
           - FALSE: Approach from negative direction (default)
           - TRUE: Approach from positive direction (after over-travel) *)
        ApproachingPositive := bApproachFromPositive;

        IF bApproachFromPositive THEN
            fbMoveVelocity(
                Axis := Axis,
                Execute := TRUE,
                Velocity := ApproachVelocity,
                Direction := MC_Positive_Direction
            );
        ELSE
            fbMoveVelocity(
                Axis := Axis,
                Execute := TRUE,
                Velocity := ApproachVelocity,
                Direction := MC_Negative_Direction
            );
        END_IF

        InMotion := fbMoveVelocity.Busy;

        IF LimitHomeActive THEN
            (* Home limit switch triggered - stop and detect *)
            fbMoveVelocity(Execute := FALSE);
            eState := HL_DETECT;

        ELSIF LimitRetractActive THEN
            (* Over-travel: Hit retract limit instead of home limit *)
            IF NOT bApproachFromPositive THEN
                (* Was approaching from negative - reverse to positive direction *)
                fbMoveVelocity(Execute := FALSE);
                bApproachFromPositive := TRUE;
                (* Stay in HL_APPROACH, will re-enter with new direction next scan *)

            ELSE
                (* Already approaching from positive and hit retract - fault *)
                fbMoveVelocity(Execute := FALSE);
                Error := TRUE;
                ErrorID := ERR_LIMIT_INVALID;
                eState := HL_ERROR;
            END_IF

        ELSIF fbMoveVelocity.Error THEN
            fbMoveVelocity(Execute := FALSE);
            Error := TRUE;
            ErrorID := ERR_DRIVE;
            eState := HL_ERROR;
        END_IF

    HL_DETECT:
        (* Halt motion after limit switch detected *)
        fbHalt(
            Axis := Axis,
            Execute := TRUE
        );

        InMotion := NOT fbHalt.Done;

        IF fbHalt.Done THEN
            fbHalt(Execute := FALSE);
            eState := HL_BACKOFF;

        ELSIF fbHalt.Error THEN
            fbHalt(Execute := FALSE);
            Error := TRUE;
            ErrorID := ERR_DRIVE;
            eState := HL_ERROR;
        END_IF

    HL_BACKOFF:
        (* Move away from limit switch at slow speed until switch clears *)
        fbMoveVelocity(
            Axis := Axis,
            Execute := TRUE,
            Velocity := BackoffVelocity,
            Direction := MC_Positive_Direction
        );

        InMotion := fbMoveVelocity.Busy;

        IF NOT LimitHomeActive THEN
            (* Switch cleared - halt and set position *)
            fbMoveVelocity(Execute := FALSE);
            eState := HL_SETREF;

        ELSIF fbMoveVelocity.Error THEN
            fbMoveVelocity(Execute := FALSE);
            Error := TRUE;
            ErrorID := ERR_DRIVE;
            eState := HL_ERROR;
        END_IF

    HL_SETREF:
        (* Set position reference at home switch edge location *)
        (* First halt to ensure fully stopped *)
        fbHalt(
            Axis := Axis,
            Execute := NOT fbHalt.Done
        );

        IF fbHalt.Done THEN
            fbHalt(Execute := FALSE);

            (* Set this position as the home reference *)
            fbSetPosition(
                Axis := Axis,
                Execute := TRUE,
                Position := SetPosition
            );

            IF fbSetPosition.Done THEN
                fbSetPosition(Execute := FALSE);
                InMotion := FALSE;
                Done := TRUE;
                eState := HL_DONE;

            ELSIF fbSetPosition.Error THEN
                fbSetPosition(Execute := FALSE);
                Error := TRUE;
                ErrorID := ERR_SETPOS;
                eState := HL_ERROR;
            END_IF
        END_IF

    HL_DONE:
        (* Homing sequence complete *)
        Done := TRUE;
        Active := TRUE;
        InMotion := FALSE;
        ApproachingPositive := FALSE;

        (* Reset when Execute goes low *)
        IF NOT Execute THEN
            Done := FALSE;
            eState := HL_IDLE;
        END_IF

    HL_ABORTING:
        (* Aborting sequence - halt motion *)
        fbHalt(
            Axis := Axis,
            Execute := TRUE
        );

        IF fbHalt.Done THEN
            fbHalt(Execute := FALSE);
            Active := FALSE;
            InMotion := FALSE;
            eState := HL_IDLE;

        ELSIF fbHalt.Error THEN
            (* Halt failed - still try to go to idle *)
            fbHalt(Execute := FALSE);
            eState := HL_ERROR;
        END_IF

    HL_ERROR:
        (* Error state *)
        Active := FALSE;
        InMotion := FALSE;
        Done := FALSE;

        (* Allow reset when Execute goes low *)
        IF NOT Execute THEN
            Error := FALSE;
            ErrorID := 0;
            eState := HL_IDLE;
        END_IF

END_CASE

END_FUNCTION_BLOCK

(* ---- FB_ModeDecoder.st ---- *)
(* ============================================================================
   FB_ModeDecoder - Mode Command Decoder

   Project: Gen3 SOS Compressor Servo Controller
   Controller: Yaskawa MP2600iec

   Description:
   Decodes the 3-bit mode command from digital inputs (DI0, DI1, DI2) into
   an E_OperatingMode enumeration value.

   NOTE: Input debouncing is handled externally by FB_DigitalInputFilter.
   This function block expects pre-filtered (debounced) inputs.

   Inputs:
   - ModeBit0, ModeBit1, ModeBit2: Filtered digital input states

   Outputs:
   - DecodedMode: The operating mode enumeration
   - ModeValue: The numeric mode value (0-7)
   - ModeStable: TRUE when all input bits have the same value as previous scan
   ============================================================================ *)

FUNCTION_BLOCK FB_ModeDecoder
VAR_INPUT
    Enable          : BOOL;             (* Enable the decoder *)
    ModeBit0        : BOOL;             (* Mode bit 0 - LSB (DI0) - pre-filtered *)
    ModeBit1        : BOOL;             (* Mode bit 1 (DI1) - pre-filtered *)
    ModeBit2        : BOOL;             (* Mode bit 2 - MSB (DI2) - pre-filtered *)
END_VAR

VAR_OUTPUT
    DecodedMode     : E_OperatingMode;  (* Decoded operating mode *)
    ModeValue       : INT;              (* Numeric mode value 0-7 *)
    ModeStable      : BOOL;             (* Mode has been stable (no change from last scan) *)
    ModeChanged     : BOOL;             (* Rising edge - mode just changed *)
END_VAR

VAR
    nCurrentValue   : INT;              (* Current mode value *)
    nPreviousValue  : INT;              (* Previous scan mode value *)
    bPrevStable     : BOOL;             (* Previous stable state *)
END_VAR

(* ============================================================================
   Main Logic
   ============================================================================ *)

IF NOT Enable THEN
    (* Reset outputs when disabled *)
    DecodedMode := MODE_IDLE;
    ModeValue := 0;
    ModeStable := FALSE;
    ModeChanged := FALSE;
    nPreviousValue := 0;
    RETURN;
END_IF

(* Decode mode from bits using centralized conversion function *)
DecodedMode := BitsToMode(ModeBit0, ModeBit1, ModeBit2);
nCurrentValue := ModeToInt(DecodedMode);

(* Update outputs *)
ModeValue := nCurrentValue;

(* Mode is stable if value matches previous scan *)
ModeStable := (nCurrentValue = nPreviousValue);

(* Detect mode change (value different from previous scan) *)
ModeChanged := (nCurrentValue <> nPreviousValue);

(* Save for next scan *)
nPreviousValue := nCurrentValue;
bPrevStable := ModeStable;

END_FUNCTION_BLOCK

(* ---- FB_OutputMux.st ---- *)
(* ============================================================================
   FB_OutputMux - Digital Output Multiplexer

   Project: Gen3 SOS Compressor Servo Controller
   Controller: Yaskawa MP2600iec

   Description:
   Multiplexes DO0-DO2 outputs between mode confirmation and fault code:
   - Normal mode: DO0-DO2 = Mode confirmation bits
   - Fault mode:  DO0-DO2 = Fault code bits

   Uses centralized conversion functions from EnumConversions.st

   Output Multiplexing:
   - Normal mode: DO0-DO2 = Mode confirmation bits (000-111)
   - Fault mode:  DO0-DO2 = Fault code bits (000-111)

   Fault Codes (3-bit):
   000 = No fault / cleared
   001 = Handshake timeout/mismatch
   010 = Drive fault
   011 = Position limit exceeded
   100 = Homing requirement not met
   101 = Piston exit prevention triggered
   110 = Limit switch fault
   111 = Encoder/absolute position fault
   ============================================================================ *)

FUNCTION_BLOCK FB_OutputMux
VAR_INPUT
    Enable              : BOOL;             (* Enable the function block *)
    FaultActive         : BOOL;             (* Fault state is active *)
    FaultCode           : E_FaultCode;      (* Current fault code *)
    ModeConfirmBit0     : BOOL;             (* Mode confirmation bit 0 *)
    ModeConfirmBit1     : BOOL;             (* Mode confirmation bit 1 *)
    ModeConfirmBit2     : BOOL;             (* Mode confirmation bit 2 *)
END_VAR

VAR_OUTPUT
    DO0_Output          : BOOL;             (* Output for DO0 *)
    DO1_Output          : BOOL;             (* Output for DO1 *)
    DO2_Output          : BOOL;             (* Output for DO2 *)
    FaultActiveOutput   : BOOL;             (* Output for doFaultActive (DO5) *)
END_VAR

VAR
    bFaultBit0          : BOOL;             (* Fault code bit 0 *)
    bFaultBit1          : BOOL;             (* Fault code bit 1 *)
    bFaultBit2          : BOOL;             (* Fault code bit 2 *)
END_VAR

(* ============================================================================
   Main Logic
   ============================================================================ *)

IF NOT Enable THEN
    (* All outputs low when disabled *)
    DO0_Output := FALSE;
    DO1_Output := FALSE;
    DO2_Output := FALSE;
    FaultActiveOutput := FALSE;
    RETURN;
END_IF

(* Set fault active output *)
FaultActiveOutput := FaultActive;

IF FaultActive THEN
    (* Fault mode: Output fault code on DO0-DO2 *)
    (* Use centralized conversion function *)
    FaultToBits(FaultCode, bFaultBit0, bFaultBit1, bFaultBit2);

    DO0_Output := bFaultBit0;
    DO1_Output := bFaultBit1;
    DO2_Output := bFaultBit2;
ELSE
    (* Normal mode: Output mode confirmation bits *)
    DO0_Output := ModeConfirmBit0;
    DO1_Output := ModeConfirmBit1;
    DO2_Output := ModeConfirmBit2;
END_IF

END_FUNCTION_BLOCK

(* ---- FB_PistonExitGuard.st ---- *)
(* ============================================================================
   FB_PistonExitGuard - Piston Exit Prevention Guard (Simplified)

   Project: Gen3 SOS Compressor Servo Controller
   Controller: Yaskawa MP2600iec

   Description:
   Monitors for dangerous condition where external pressure is pushing the
   piston out of the cylinder despite motor resistance. This is a DETECTION-ONLY
   function block - it does NOT modify commands, only triggers a fault when
   the dangerous condition is detected.

   The cylinder contains pressurized oxygen micro-bubble solution. If the piston
   exits the cylinder while pressurized, dangerous spray would result.

   SIGN CONVENTION (CRITICAL):
   - Positive direction: Toward cylinder EOT (compression, INTO cylinder)
   - Negative direction: Toward exit (retract, OUT OF cylinder)
   - Pressure pushes piston OUT (negative direction)
   - Motor RESISTS with POSITIVE torque to hold piston IN

   DANGEROUS CONDITION:
   When near the exit boundary, if:
   - Motor is applying positive torque (resisting/pushing into cylinder)
   - But actual velocity is negative (moving toward exit anyway)
   Then external pressure is overcoming motor resistance - FAULT!

   Integration:
   - Called from PRG_Main safety monitoring section
   - FaultTriggered connects to FB_SafetyMonitor.ExitGuardTriggered
   - Caller is responsible for transitioning to ST_FAULT when triggered
   ============================================================================ *)

FUNCTION_BLOCK FB_PistonExitGuard
VAR_INPUT
    Enable              : BOOL;             (* Enable the guard *)

    (* Axis state - actual values only *)
    ActualPosition      : LREAL;            (* Current position (mm) *)
    ActualVelocity      : LREAL;            (* Current velocity (mm/s) *)
    ActualTorque        : LREAL;            (* Current torque (%) *)

    (* Limit configuration *)
    SoftLimitMin        : LREAL;            (* Minimum allowed position (mm) *)
    GuardMargin         : LREAL;            (* Safety margin before limit (mm) *)

    (* Detection thresholds *)
    VelocityThreshold   : LREAL;            (* Motion detection threshold (mm/s) *)
    TorqueThreshold     : LREAL;            (* Torque threshold for detection (%) *)
END_VAR

VAR_OUTPUT
    (* Status outputs *)
    FaultTriggered      : BOOL;             (* Dangerous condition detected - transition to fault *)
    GuardActive         : BOOL;             (* Guard is actively monitoring *)

    (* Diagnostic outputs *)
    InDangerZone        : BOOL;             (* Position is near exit limit *)
    ApproachingLimit    : BOOL;             (* Moving toward exit limit *)
END_VAR

VAR
    rGuardBoundary      : LREAL;            (* Boundary = SoftLimitMin + GuardMargin *)
END_VAR

(* ============================================================================
   Main Logic
   ============================================================================ *)

IF NOT Enable THEN
    (* Reset all outputs when disabled *)
    FaultTriggered := FALSE;
    GuardActive := FALSE;
    InDangerZone := FALSE;
    ApproachingLimit := FALSE;
    RETURN;
END_IF

(* Calculate guard boundary *)
rGuardBoundary := SoftLimitMin + GuardMargin;

(* Determine position and motion status *)
InDangerZone := (ActualPosition <= rGuardBoundary);
ApproachingLimit := (ActualVelocity < -VelocityThreshold);  (* Negative = toward exit *)

(* Guard is always active when enabled *)
GuardActive := TRUE;

(* Reset fault before evaluation *)
FaultTriggered := FALSE;

(* --------------------------------------------------------------------------
   DANGEROUS CONDITION DETECTION

   Detect: Near exit + positive torque (resisting) + negative velocity (moving out)

   This indicates external pressure is pushing the piston out despite the motor
   applying resistance (positive torque). The motor is trying to hold/push the
   piston into the cylinder but the pressure is winning.

   Sign convention:
   - Positive torque = motor pushing INTO cylinder (resisting exit)
   - Negative velocity = piston moving OUT of cylinder (toward exit)
   - Both together near exit = pressure overcoming motor = DANGER
   -------------------------------------------------------------------------- *)

IF InDangerZone THEN
    (* In danger zone - check for anomalous pressure condition *)

    IF (ActualTorque > TorqueThreshold) AND          (* Motor applying positive torque - resisting *)
       (ActualVelocity < -VelocityThreshold) THEN    (* But still moving toward exit *)
        (* DANGEROUS: Pressure overcoming motor resistance *)
        FaultTriggered := TRUE;
    END_IF
END_IF

(* --------------------------------------------------------------------------
   HARD LIMIT VIOLATION

   If position has gone below absolute minimum, always fault regardless of
   torque/velocity. This is a backup check.
   -------------------------------------------------------------------------- *)

IF ActualPosition < SoftLimitMin THEN
    FaultTriggered := TRUE;
END_IF

END_FUNCTION_BLOCK

(* ---- FB_PositionOutput.st ---- *)
(* ============================================================================
   FB_PositionOutput - Two-Stage Position Output Signal Mapping

   Project: Gen3 SOS Compressor Servo Controller
   Controller: Yaskawa MP2600iec

   Description:
   Maps the actual position to analog output voltage using a two-stage
   scaling scheme for improved resolution in the critical in-cylinder region.
   This signal is sent to the master controller.

   Two-Stage Mapping:
   - Stage 1: In-cylinder region (higher resolution)
     Position 0-200mm maps to -10V to +5V (15V range for 200mm)
   - Stage 2: Out-of-cylinder region (lower resolution)
     Position 200-305mm maps to +5V to +10V (5V range for 105mm)

   This provides approximately 3x better resolution in the working region
   where the piston is inside the cylinder.

   Output:
   - Raw INT: -32768 to +32767 corresponds to -10V to +10V
   ============================================================================ *)

FUNCTION_BLOCK FB_PositionOutput
VAR_INPUT
    Enable              : BOOL;             (* Enable the mapper *)
    ActualPosition      : LREAL;            (* Current position in mm *)

    (* Stage 1 configuration (in-cylinder, higher resolution) *)
    Stage1PosMin        : LREAL;            (* Stage 1 position start (mm) *)
    Stage1PosMax        : LREAL;            (* Stage 1 position end (mm) *)
    Stage1VoltMin       : LREAL;            (* Stage 1 voltage start (V) *)
    Stage1VoltMax       : LREAL;            (* Stage 1 voltage end (V) *)

    (* Stage 2 configuration (out-of-cylinder, lower resolution) *)
    Stage2PosMin        : LREAL;            (* Stage 2 position start (mm) *)
    Stage2PosMax        : LREAL;            (* Stage 2 position end (mm) *)
    Stage2VoltMin       : LREAL;            (* Stage 2 voltage start (V) *)
    Stage2VoltMax       : LREAL;            (* Stage 2 voltage end (V) *)
END_VAR

VAR_OUTPUT
    RawAnalogOutput     : INT;              (* Raw analog output value *)
    OutputVoltage       : LREAL;            (* Calculated output voltage *)
    InStage1            : BOOL;             (* Position is in stage 1 region *)
    InStage2            : BOOL;             (* Position is in stage 2 region *)
END_VAR

VAR
    rVoltage            : LREAL;            (* Calculated voltage *)
    rNormalized         : LREAL;            (* Normalized position within stage *)
    rRawValue           : LREAL;            (* Raw value before conversion *)
END_VAR

(* ============================================================================
   Constants
   ============================================================================ *)
VAR CONSTANT
    RAW_MIN             : LREAL := -32768.0;    (* Minimum raw value *)
    RAW_MAX             : LREAL := 32767.0;     (* Maximum raw value *)
    VOLT_MIN            : LREAL := -10.0;       (* Minimum voltage *)
    VOLT_MAX            : LREAL := 10.0;        (* Maximum voltage *)
    VOLT_RANGE          : LREAL := 20.0;        (* Total voltage range *)
END_VAR

(* ============================================================================
   Main Logic
   ============================================================================ *)

IF NOT Enable THEN
    RawAnalogOutput := 0;
    OutputVoltage := 0.0;
    InStage1 := FALSE;
    InStage2 := FALSE;
    RETURN;
END_IF

(* Determine which stage the position falls into *)
IF ActualPosition <= Stage1PosMax THEN
    (* Stage 1: In-cylinder region *)
    InStage1 := TRUE;
    InStage2 := FALSE;

    (* Calculate normalized position within stage 1 *)
    IF (Stage1PosMax - Stage1PosMin) > 0.0 THEN
        rNormalized := (ActualPosition - Stage1PosMin) / (Stage1PosMax - Stage1PosMin);
    ELSE
        rNormalized := 0.0;
    END_IF

    (* Clamp to 0.0-1.0 range *)
    rNormalized := LIMIT(0.0, rNormalized, 1.0);

    (* Calculate voltage for stage 1 *)
    rVoltage := Stage1VoltMin + (rNormalized * (Stage1VoltMax - Stage1VoltMin));

ELSE
    (* Stage 2: Out-of-cylinder region *)
    InStage1 := FALSE;
    InStage2 := TRUE;

    (* Calculate normalized position within stage 2 *)
    IF (Stage2PosMax - Stage2PosMin) > 0.0 THEN
        rNormalized := (ActualPosition - Stage2PosMin) / (Stage2PosMax - Stage2PosMin);
    ELSE
        rNormalized := 0.0;
    END_IF

    (* Clamp to 0.0-1.0 range *)
    rNormalized := LIMIT(0.0, rNormalized, 1.0);

    (* Calculate voltage for stage 2 *)
    rVoltage := Stage2VoltMin + (rNormalized * (Stage2VoltMax - Stage2VoltMin));
END_IF

(* Clamp voltage to valid range *)
rVoltage := LIMIT(VOLT_MIN, rVoltage, VOLT_MAX);
OutputVoltage := rVoltage;

(* Convert voltage to raw output value *)
(* Voltage -10V to +10V maps to raw -32768 to +32767 *)
rRawValue := ((rVoltage - VOLT_MIN) / VOLT_RANGE) * (RAW_MAX - RAW_MIN) + RAW_MIN;

(* Convert to integer with clamping *)
IF rRawValue < RAW_MIN THEN
    RawAnalogOutput := -32768;
ELSIF rRawValue > RAW_MAX THEN
    RawAnalogOutput := 32767;
ELSE
    RawAnalogOutput := LREAL_TO_INT(rRawValue);
END_IF

END_FUNCTION_BLOCK

(* ---- FB_SafetyMonitor.st ---- *)
(* ============================================================================
   FB_SafetyMonitor - Centralized Safety Monitoring

   Project: Gen3 SOS Compressor Servo Controller
   Controller: Yaskawa MP2600iec

   Description:
   Monitors all safety-related conditions and generates appropriate fault codes.
   This function block provides a single point for all safety monitoring,
   making the system easier to audit and maintain.

   Monitored Conditions:
   - Drive faults (from servo amplifier)
   - Encoder faults (invalid position, battery low)
   - Limit switch faults (unexpected triggers during motion)
   - Position limit violations (beyond soft limits)
   - Piston exit guard faults (from FB_PistonExitGuard)

   Fault Priority (highest to lowest):
   1. Drive fault (FAULT_DRIVE)
   2. Encoder fault (FAULT_ENCODER)
   3. Limit switch fault (FAULT_LIMIT_SWITCH)
   4. Position limit fault (FAULT_POSITION)
   5. Piston exit fault (FAULT_PISTON_EXIT)

   Integration:
   - Called every scan after state machine, before output update
   - FaultDetected triggers transition to ST_FAULT in PRG_Main
   ============================================================================ *)

FUNCTION_BLOCK FB_SafetyMonitor
VAR_INPUT
    Enable              : BOOL;             (* Enable safety monitoring *)

    (* Limit switch status - from filtered digital inputs *)
    LimitRetractActive  : BOOL;             (* TRUE = retract limit triggered *)
    LimitHomeActive     : BOOL;             (* TRUE = home limit triggered *)

    (* Position information *)
    ActualPosition      : LREAL;            (* Current axis position (mm) *)
    SoftLimitMin        : LREAL;            (* Minimum allowed position (mm) *)
    SoftLimitMax        : LREAL;            (* Maximum allowed position (mm) *)

    (* Drive status *)
    DriveReady          : BOOL;             (* Drive is ready for motion *)
    DriveFault          : BOOL;             (* Drive has reported a fault *)
    DriveErrorID        : DWORD;            (* Drive error code if fault *)

    (* Encoder status *)
    EncoderValid        : BOOL;             (* Absolute encoder position valid *)
    EncoderBatteryOK    : BOOL;             (* Encoder battery status OK *)

    (* Operating context *)
    CurrentState        : E_SystemState;    (* Current state machine state *)
    CurrentMode         : E_OperatingMode;  (* Current operating mode *)

    (* Piston exit guard status *)
    ExitGuardTriggered  : BOOL;             (* Piston exit guard triggered fault *)
END_VAR

VAR_OUTPUT
    (* Primary fault output *)
    FaultDetected       : BOOL;             (* A fault condition exists *)
    FaultCode           : E_FaultCode;      (* Fault code to report *)

    (* Individual fault flags for diagnostics *)
    FaultLimitSwitch    : BOOL;             (* Limit switch fault detected *)
    FaultPosition       : BOOL;             (* Position limit exceeded *)
    FaultDrive          : BOOL;             (* Drive fault detected *)
    FaultEncoder        : BOOL;             (* Encoder fault detected *)
    FaultPistonExit     : BOOL;             (* Piston exit guard fault *)
END_VAR

VAR
    (* Latching for fault persistence *)
    bLatchedFault       : BOOL;
    eLatchedFaultCode   : E_FaultCode;

    (* Internal flags *)
    bInMotionState      : BOOL;
    bInHomingState      : BOOL;
    bInFaultState       : BOOL;
END_VAR

(* ============================================================================
   Main Logic
   ============================================================================ *)

IF NOT Enable THEN
    (* Reset all outputs when disabled *)
    FaultDetected := FALSE;
    FaultCode := FAULT_NONE;
    FaultLimitSwitch := FALSE;
    FaultPosition := FALSE;
    FaultDrive := FALSE;
    FaultEncoder := FALSE;
    FaultPistonExit := FALSE;
    bLatchedFault := FALSE;
    eLatchedFaultCode := FAULT_NONE;
    RETURN;
END_IF

(* --------------------------------------------------------------------------
   Determine operating context
   -------------------------------------------------------------------------- *)

(* Check if in a motion state *)
bInMotionState := (CurrentState = ST_POSITION_CTRL) OR
                  (CurrentState = ST_VELOCITY_CTRL) OR
                  (CurrentState = ST_TORQUE_CTRL) OR
                  (CurrentState = ST_GO_HOME) OR
                  (CurrentState = ST_HOLD_POSITION);

(* Check if in a homing state *)
bInHomingState := (CurrentState = ST_HOME_LIMIT) OR
                  (CurrentState = ST_HOME_LIM_APPROACH) OR
                  (CurrentState = ST_HOME_LIM_DETECT) OR
                  (CurrentState = ST_HOME_LIM_BACKOFF) OR
                  (CurrentState = ST_HOME_LIM_SETREF) OR
                  (CurrentState = ST_HOME_EOT) OR
                  (CurrentState = ST_HOME_EOT_FAST) OR
                  (CurrentState = ST_HOME_EOT_SLOW) OR
                  (CurrentState = ST_HOME_EOT_DETECT) OR
                  (CurrentState = ST_HOME_EOT_SETREF) OR
                  (CurrentState = ST_HOME_COMPLETE);

(* Check if already in fault state *)
bInFaultState := (CurrentState = ST_FAULT) OR
                 (CurrentState = ST_FAULT_RECOVERY) OR
                 (CurrentState = ST_FAULT_IDLE);

(* --------------------------------------------------------------------------
   Reset fault latch when appropriate
   -------------------------------------------------------------------------- *)

(* Clear fault latch when entering fault idle or returning to idle *)
IF (CurrentState = ST_FAULT_IDLE) OR (CurrentState = ST_IDLE) THEN
    IF NOT FaultDetected THEN
        bLatchedFault := FALSE;
        eLatchedFaultCode := FAULT_NONE;
    END_IF
END_IF

(* --------------------------------------------------------------------------
   DRIVE FAULT MONITORING
   Most critical - servo amplifier has detected an issue
   -------------------------------------------------------------------------- *)

FaultDrive := DriveFault;

(* --------------------------------------------------------------------------
   ENCODER FAULT MONITORING
   Invalid position data or battery issues
   -------------------------------------------------------------------------- *)

(* Encoder is faulty if position invalid (but only check when relevant) *)
(* Don't trigger encoder fault during initialization before check completes *)
IF (CurrentState > ST_ENCODER_CHECK) THEN
    FaultEncoder := NOT EncoderValid;
ELSE
    FaultEncoder := FALSE;
END_IF

(* --------------------------------------------------------------------------
   LIMIT SWITCH FAULT MONITORING
   Unexpected limit switch activation during motion
   -------------------------------------------------------------------------- *)

(* Limit switches are expected during homing - only fault if unexpected *)
IF bInMotionState AND NOT bInHomingState THEN
    (* During normal motion, hitting a limit switch is unexpected *)
    (* This could indicate mechanical issue, runaway, or position error *)
    IF LimitRetractActive OR LimitHomeActive THEN
        FaultLimitSwitch := TRUE;
    ELSE
        FaultLimitSwitch := FALSE;
    END_IF
ELSE
    (* Not in motion or in homing - limits are OK or expected *)
    FaultLimitSwitch := FALSE;
END_IF

(* --------------------------------------------------------------------------
   POSITION LIMIT MONITORING
   Position beyond software limits
   -------------------------------------------------------------------------- *)

(* Check if position is outside software limits *)
IF (ActualPosition < SoftLimitMin) OR (ActualPosition > SoftLimitMax) THEN
    FaultPosition := TRUE;
ELSE
    FaultPosition := FALSE;
END_IF

(* --------------------------------------------------------------------------
   PISTON EXIT GUARD MONITORING
   Triggered by FB_PistonExitGuard
   -------------------------------------------------------------------------- *)

FaultPistonExit := ExitGuardTriggered;

(* --------------------------------------------------------------------------
   FAULT PRIORITY AND OUTPUT
   Determine highest priority fault and set outputs
   -------------------------------------------------------------------------- *)

(* Priority order: Drive > Encoder > LimitSwitch > Position > PistonExit *)
IF FaultDrive THEN
    FaultDetected := TRUE;
    FaultCode := FAULT_DRIVE;

ELSIF FaultEncoder THEN
    FaultDetected := TRUE;
    FaultCode := FAULT_ENCODER;

ELSIF FaultLimitSwitch THEN
    FaultDetected := TRUE;
    FaultCode := FAULT_LIMIT_SWITCH;

ELSIF FaultPosition THEN
    FaultDetected := TRUE;
    FaultCode := FAULT_POSITION;

ELSIF FaultPistonExit THEN
    FaultDetected := TRUE;
    FaultCode := FAULT_PISTON_EXIT;

ELSE
    FaultDetected := FALSE;
    FaultCode := FAULT_NONE;
END_IF

(* --------------------------------------------------------------------------
   FAULT LATCHING
   Latch fault for persistence across scans until explicitly cleared
   -------------------------------------------------------------------------- *)

IF FaultDetected AND NOT bLatchedFault AND NOT bInFaultState THEN
    bLatchedFault := TRUE;
    eLatchedFaultCode := FaultCode;
END_IF

(* Use latched fault if current scan doesn't detect new fault *)
IF bLatchedFault AND NOT FaultDetected THEN
    FaultDetected := TRUE;
    FaultCode := eLatchedFaultCode;
END_IF

END_FUNCTION_BLOCK

(* ---- FB_BitsToFaultCode.st ---- *)
(* ============================================================================
   FB_BitsToFaultCode - Convert 3 Digital Input Bits to Fault Code

   Project: Gen3 SOS Compressor Servo Controller
   Controller: Yaskawa MP2600iec

   Description:
   Converts 3 digital input bits to the corresponding E_FaultCode
   enumeration value. Used during fault reset to decode the master's
   fault acknowledgement from DI0-DI2.

   NOTE: Implemented as an FB (not an FN) to work around a MotionWorks IEC
   native-code-gen defect on FUNCTIONs with user-enum return types.

   Variables (define in MWiec GUI):
     VAR_INPUT:
       Bit0            : BOOL             (* LSB
       Bit1            : BOOL
       Bit2            : BOOL             (* MSB
     VAR_OUTPUT:
       Fault           : E_FaultCode      (* Decoded fault code
     VAR:
       nValue          : INT              (* Calculated integer value
   ============================================================================ *)

(* Calculate integer value from bits *)
nValue := 0;
IF Bit0 THEN nValue := nValue + 1; END_IF;
IF Bit1 THEN nValue := nValue + 2; END_IF;
IF Bit2 THEN nValue := nValue + 4; END_IF;

(* Convert integer to fault code *)
IF nValue = 0 THEN
    Fault := E_FaultCode#FAULT_NONE;
ELSIF nValue = 1 THEN
    Fault := E_FaultCode#FAULT_HANDSHAKE;
ELSIF nValue = 2 THEN
    Fault := E_FaultCode#FAULT_DRIVE;
ELSIF nValue = 3 THEN
    Fault := E_FaultCode#FAULT_POSITION;
ELSIF nValue = 4 THEN
    Fault := E_FaultCode#FAULT_HOMING_REQ;
ELSIF nValue = 5 THEN
    Fault := E_FaultCode#FAULT_PISTON_EXIT;
ELSIF nValue = 6 THEN
    Fault := E_FaultCode#FAULT_LIMIT_SWITCH;
ELSIF nValue = 7 THEN
    Fault := E_FaultCode#FAULT_ENCODER;
ELSE
    Fault := E_FaultCode#FAULT_NONE;
END_IF;

(* ---- FB_BitsToMode.st ---- *)
(* ============================================================================
   FB_BitsToMode - Convert 3 Digital Input Bits to Operating Mode

   Project: Gen3 SOS Compressor Servo Controller
   Controller: Yaskawa MP2600iec

   Description:
   Converts 3 digital input bits to the corresponding E_OperatingMode
   enumeration value. Calculates the integer value from bits then
   maps to the corresponding mode.

   NOTE: Implemented as an FB (not an FN) to work around a MotionWorks IEC
   native-code-gen defect on FUNCTIONs with user-enum return types.

   Variables (define in MWiec GUI):
     VAR_INPUT:
       Bit0            : BOOL             (* LSB
       Bit1            : BOOL
       Bit2            : BOOL             (* MSB
     VAR_OUTPUT:
       Mode            : E_OperatingMode  (* Decoded operating mode
     VAR:
       nValue          : INT              (* Calculated integer value
   ============================================================================ *)

(* Calculate integer value from bits *)
nValue := 0;
IF Bit0 THEN nValue := nValue + 1; END_IF;
IF Bit1 THEN nValue := nValue + 2; END_IF;
IF Bit2 THEN nValue := nValue + 4; END_IF;

(* Convert integer to mode *)
IF nValue = 0 THEN
    Mode := E_OperatingMode#MODE_IDLE;
ELSIF nValue = 1 THEN
    Mode := E_OperatingMode#MODE_BRAKE_HOLD;
ELSIF nValue = 2 THEN
    Mode := E_OperatingMode#MODE_POSITION;
ELSIF nValue = 3 THEN
    Mode := E_OperatingMode#MODE_VELOCITY;
ELSIF nValue = 4 THEN
    Mode := E_OperatingMode#MODE_TORQUE;
ELSIF nValue = 5 THEN
    Mode := E_OperatingMode#MODE_GO_HOME;
ELSIF nValue = 6 THEN
    Mode := E_OperatingMode#MODE_HOME_LIMIT;
ELSIF nValue = 7 THEN
    Mode := E_OperatingMode#MODE_RESERVED_111;
ELSE
    Mode := E_OperatingMode#MODE_IDLE;
END_IF;
